(* PLC project static_torsion.project, CODESYS CODESYS V3.5 SP17 Patch 3 *)
(* stored: creationDateTime 1970-01-01T00:00:00, modificationDateTime 2026-06-22T15:12:39.4699931 *)

FUNCTION _word_to_real : REAL
  VAR_INPUT
    _word2 : ARRAY[0..1] OF WORD;
  END_VAR
  VAR
    _RW : REAL_WORD2;
  END_VAR

            _RW._WORDS := _word2;
_word_to_real := _RW._REAL;
          
END_FUNCTION
